// TwinCAT 3 PLC project lcls_plc_lps_02
// Title: lcls-plc-pls-02
// Company: SLAC
// ProjectVersion: 1.0.0
// ProgramVersion: 3.1.4022.7
// libraries:
//   Tc2_BABasic, * (Beckhoff Automation GmbH)
//   Tc2_EtherCAT, * (Beckhoff Automation GmbH)
//   Tc2_ModbusRTU, * (Beckhoff Automation GmbH)
//   Tc2_Standard, * (Beckhoff Automation GmbH)
//   Tc2_System, * (Beckhoff Automation GmbH)
//   Tc3_Module, * (Beckhoff Automation GmbH)
// project tree:
//   DUTs/ E_ShutterState.TcDUT, E_DeviceState.TcDUT, E_Mode.TcDUT, E_LeakLocation.TcDUT, ST_DeviceDiagnostic.TcDUT, ST_ErrorStates.TcDUT, ST_LaserSetpoints.TcDUT, ST_LeakBoundaries.TcDUT, ST_TemperatureMonitorSetpoints.TcDUT
//   GVLs/ GVL_EL3174.TcGVL, GVL_IO.TcGVL, GVL_Laser.TcGVL, GVL_PLC.TcGVL, GVL_TemperatureMonitor.TcGVL, GVL_TraceTek.TcGVL
//   / PlcTask.TcTTO
//   POUs/Communication/ FB_TraceTekModbus.TcPOU
//   POUs/Devices/ FB_BaseplateChiller.TcPOU, FB_Amphos_Enable.TcPOU, FB_ChillerLoop.TcPOU, FB_DumpChiller.TcPOU, FB_LaserInterlock.TcPOU, FB_Laser_Timer.TcPOU, FB_Laser_Timer_MPC.TcPOU, FB_LeakMonitor.TcPOU, FB_ShutterControl.TcPOU
//   POUs/Diagnostics/ FB_EcatDiag.TcPOU
//   POUs/Helpers/ FB_ErrorTriggers.TcPOU
//   POUs/Interlocks/ F_BaseplateChillerEnable.TcPOU, F_DumpChillerEnable.TcPOU
//   POUs/ MAIN.TcPOU
// real-time tasks:
//   TASK PlcTask: cycle T#10ms, priority 20, ADS port 350
// I/O:
//   DEVICE Device 1 (EtherCAT), AmsNetId 172.21.160.71.2.1
//     B950-231B-R03-DRL-01 (EK1200) [EK1200-5000 EtherCAT Power supply (2A E-Bus)]
//       EL3174_00_01 [EL3174 4Ch. Ana. Input +/-10V Diff., +/-20mA SingleEnded, 16 Bit]
//       EL3174_00_02 [EL3174 4Ch. Ana. Input +/-10V Diff., +/-20mA SingleEnded, 16 Bit]
//       EL9189_00_03 [EL9189 Potential Connection, 16 x Ground]
//       EL1259_00_04 [EL1259 8Ch. Dig Input 24V/8Ch. Dig. Output 24V with Multi-Time-Stamp]
//       EL9184_00_05 [EL9184 Potential Connection, 8 x 24V, 8 x Ground]
//       EL2624_00_07 [EL2624 4Ch. Relay Output, NO (125V AC / 30V DC)]
//       EL2624_00_08 [EL2624 4Ch. Relay Output, NO (125V AC / 30V DC)]
//       EL1004_00_8A
//       EL6022_00_09 [EL6022 Interface 2Ch. (RS422/485)]
//       EL9505_00_10
//       EL1124_00_11 [EL1124 4Ch. Dig. Input 5V, 10µs, Sensor Power]
//       EL1124_00_12
//       EL9011_00_12 [EL9011 End Terminal]
// variable links:
//   lcls_plc_lps_02 Instance <-> Device 1 (EtherCAT)/B950-231B-R03-DRL-01 (EK1200)/EL1004_00_8A
//     PlcTask Inputs/GVL_IO.bMirrorStatus <-> Channel 1/Input
//   lcls_plc_lps_02 Instance <-> Device 1 (EtherCAT)/B950-231B-R03-DRL-01 (EK1200)/EL1124_00_11
//     PlcTask Inputs/GVL_IO.bAmphosLaserReady <-> Channel 4/Input
//     PlcTask Inputs/GVL_IO.bAmphosOn <-> Channel 1/Input
//     PlcTask Inputs/GVL_IO.bAmphosShutterStatus <-> Channel 2/Input
//     PlcTask Inputs/GVL_IO.bCarbideOn <-> Channel 3/Input
//   lcls_plc_lps_02 Instance <-> Device 1 (EtherCAT)/B950-231B-R03-DRL-01 (EK1200)/EL1124_00_12
//     PlcTask Inputs/GVL_IO.bAmphosLaserACK <-> Channel 1/Input
//     PlcTask Inputs/GVL_IO.bAmphosLaserBusy <-> Channel 2/Input
//   lcls_plc_lps_02 Instance <-> Device 1 (EtherCAT)/B950-231B-R03-DRL-01 (EK1200)/EL1259_00_04
//     PlcTask Inputs/GVL_IO.bBaseplateChillerFlow <-> MTI Inputs 10x Channel 8/Status/Input state
//     PlcTask Inputs/GVL_IO.bDumpChillerFlow <-> MTI Inputs 10x Channel 7/Status/Input state
//     PlcTask Inputs/GVL_IO.bLoopTempSW01 <-> MTI Inputs 10x Channel 3/Status/Input state
//     PlcTask Inputs/GVL_IO.bLoopTempSW02 <-> MTI Inputs 10x Channel 4/Status/Input state
//     PlcTask Inputs/GVL_IO.bLoopTempSW03 <-> MTI Inputs 10x Channel 5/Status/Input state
//     PlcTask Inputs/GVL_IO.bLoopTempSW04 <-> MTI Inputs 10x Channel 6/Status/Input state
//     PlcTask Inputs/GVL_IO.bLoopTempSW05 <-> MTI Inputs 10x Channel 1/Status/Input state
//     PlcTask Inputs/GVL_IO.bTracetekAlarm <-> MTI Inputs 10x Channel 2/Status/Input state
//   lcls_plc_lps_02 Instance <-> Device 1 (EtherCAT)/B950-231B-R03-DRL-01 (EK1200)/EL2624_00_07
//     PlcTask Outputs/GVL_IO.bAmphosEnable <-> Channel 3/Output
//     PlcTask Outputs/GVL_IO.bBaseplateChillerRelay <-> Channel 2/Output
//     PlcTask Outputs/GVL_IO.bCarbideShutterEnable <-> Channel 4/Output
//     PlcTask Outputs/GVL_IO.bDumpChillerRelay <-> Channel 1/Output
//   lcls_plc_lps_02 Instance <-> Device 1 (EtherCAT)/B950-231B-R03-DRL-01 (EK1200)/EL2624_00_08
//     PlcTask Outputs/GVL_IO.bAmphosRelayCLOSE <-> Channel 4/Output
//     PlcTask Outputs/GVL_IO.bAmphosRelayOPEN <-> Channel 1/Output
//   lcls_plc_lps_02 Instance <-> Device 1 (EtherCAT)/B950-231B-R03-DRL-01 (EK1200)/EL3174_00_01
//     PlcTask Inputs/GVL_IO.nMultiPassVoltageRaw <-> AI Standard Channel 3/Value
//     PlcTask Inputs/GVL_IO.nOpcpaVoltageRaw <-> AI Standard Channel 1/Value
//   lcls_plc_lps_02 Instance <-> Device 1 (EtherCAT)/B950-231B-R03-DRL-01 (EK1200)/EL3174_00_02
//     PlcTask Inputs/GVL_IO.nAmphosVoltageRaw <-> AI Standard Channel 1/Value
//   lcls_plc_lps_02 Instance <-> Device 1 (EtherCAT)/B950-231B-R03-DRL-01 (EK1200)/EL6022_00_09
//     PlcTask Inputs/MAIN.fbTraceTekModbus.fbModbusMaster.InData/D <-> COM Inputs Channel 2/Data In 0
//     PlcTask Inputs/MAIN.fbTraceTekModbus.fbModbusMaster.InData/D @bit {8..168 step 8} <-> COM Inputs Channel 2/Data In {1..21}  (21 links)
//     PlcTask Inputs/MAIN.fbTraceTekModbus.fbModbusMaster.InData/Status <-> COM Inputs Channel 2/Status
//     PlcTask Outputs/MAIN.fbTraceTekModbus.fbModbusMaster.OutData/Ctrl <-> COM Outputs Channel 2/Ctrl
//     PlcTask Outputs/MAIN.fbTraceTekModbus.fbModbusMaster.OutData/D <-> COM Outputs Channel 2/Data Out 0
//     PlcTask Outputs/MAIN.fbTraceTekModbus.fbModbusMaster.OutData/D @bit {8..168 step 8} <-> COM Outputs Channel 2/Data Out {1..21}  (21 links)

CONFIGURATION lcls_plc_lps_02
    RESOURCE PLC ON TwinCAT3
        TASK PlcTask(INTERVAL := T#10ms, PRIORITY := 20);
        PROGRAM MAIN WITH PlcTask : MAIN;
    END_RESOURCE
END_CONFIGURATION

// ---- DUTs/E_ShutterState.TcDUT
{attribute 'qualified_only'}
{attribute 'strict'}
TYPE E_ShutterState :
(
    INIT := 0 ,
    OPENREQ := 1,
    OPENACK := 2,
    OPENTOGGLE := 3,
    OPENREADY:= 4,
    OPENED := 5,
    CLOSEREQ := 6,
    CLOSEACK := 7,
    CLOSETOGGLE := 8,
    CLOSEREADY := 9,
    CLOSED := 10,
    AMPHOSOFF := 11
);
END_TYPE

// ---- DUTs/E_DeviceState.TcDUT
{attribute 'qualified_only'}
TYPE E_DeviceState :
(
    INVALID := 0,
    INIT := EC_DEVICE_STATE_INIT,
    PREOP := EC_DEVICE_STATE_PREOP,
    BOOTSTRAP := EC_DEVICE_STATE_BOOTSTRAP,
    SAFEOP := EC_DEVICE_STATE_SAFEOP,
    OP := EC_DEVICE_STATE_OP
) WORD := INVALID;
END_TYPE

// ---- DUTs/E_Mode.TcDUT
{attribute 'qualified_only'}
TYPE E_Mode :
(
    MASTER_Override :=1,
    Protection := 2,
    AMPHOS_Maintenance := 3
);
END_TYPE

// ---- DUTs/E_LeakLocation.TcDUT
{attribute 'qualified_only'}
{attribute 'strict'}
TYPE E_LeakLocation :
(
    NO_LEAK := 0,
    LOC1 := 1,
    LOC2 := 2,
    LOC3 := 4,
    LOC4 := 8,
    LOC5 := 16,
    LOC6 := 32
) BYTE;
END_TYPE

// ---- DUTs/ST_DeviceDiagnostic.TcDUT
// PLC Terminal device diagnostics
TYPE ST_DeviceDiagnostic :
STRUCT
    {attribute 'pytmc' := '
        pv: TYPE
        io: i
    '}
    sType : STRING[15];
    {attribute 'pytmc' := '
        pv: ADDRESS
        io: i
    '}
    nAddr : WORD;
    {attribute 'pytmc' := '
        pv: NAME
        io: i
    '}
    sName : STRING[31];
    {attribute 'pytmc' := '
        pv: DEVICE_STATE
        io: i
        field: ZRVL 0
        field: ONVL 1
        field: TWVL 2
        field: THVL 3
        field: FRVL 4
        field: SXVL	8
        field: ZRST INVALID
        field: ONST INIT
        field: TWST PREOP
        field: THST BOOTSTRAP
        field: FRST SAFEOP
        field: SXST OP
        field: ZRSV MAJOR
        field: ONSV MAJOR
        field: TWSV MAJOR
        field: THSV MAJOR
        field: FRSV MAJOR
        field: FVSV MINOR
        field: SXSV NO_ALARM
        field: UNSV MAJOR
    '}
    nDeviceState : ENUM;
    {attribute 'pytmc' := '
        pv: DEVICE_STATE_FLAGS
        io: i
    '}
    nDeviceStateFlags : BYTE;
    {attribute 'pytmc' := '
        pv: LINK_STATE_FLAGS
        io: i
    '}
    nLinkStateFlags : BYTE;
END_STRUCT
END_TYPE

// ---- DUTs/ST_ErrorStates.TcDUT
// Error states that can occur in the program
TYPE ST_ErrorStates :
STRUCT
    // Leak Alarms
    bLeakOpticalTableAmphosOn : BOOL; // Leak on the optical table with Amphos on
    bLeakOpticalTableNoLaser : BOOL; // Leak on the optical table with no laser on
    bLeakOpcpaCarbideOn : BOOL; // Leak inside the OPCPA with Carbide on
    bLeakUnderTable : BOOL; // Leak under the table
    bLeakInsideRacks : BOOL; // Leak inside the racks

   // Temperature loop alarms
    bChillerLoop01 : BOOL; // Temperature too high in loop 01
    bChillerLoop02 : BOOL; // Temperature too high in loop 02
    bChillerLoop03 : BOOL; // Temperature too high in loop 03
    bChillerLoop04 : BOOL; // Temperature too high in loop 04
    bChillerLoop05 : BOOL; // Temperature too high in loop 05

    // Beam Errors
    bAmphosBeam : BOOL; // Amphos beam error
    bOpcpaBeam : BOOL; // OPCPA beam error
    bMPCBeam :BOOL;    // MPC beam error

    // Temperature monitors
    bTempMon01 : BOOL; // Temperature too high at location 01
    bTempMon02 : BOOL; // Temperature too high at location 02
    bTempMon03 : BOOL; // Temperature too high at location 03
    bTempMon04 : BOOL; // Temperature too high at location 04
    bTempMon05 : BOOL; // Temperature too high at location 05
    bTempMon06 : BOOL; // Temperature too high at location 06
    bTempMon07 : BOOL; // Temperature too high at location 07
    bTempMon08 : BOOL; // Temperature too high at location 08


    // Dump chiller
    bDumpChiller : BOOL; // Dump chiller error
    bBaseplateChiller : BOOL; // Baseplate chiller error

    // Hardware Failure
    bHardwareFailure : BOOL; // A component of the EPS has failed

    //Amphos Relay
    bAmphosRelay : BOOL; // Amphos Enable error

END_STRUCT
END_TYPE

// ---- DUTs/ST_LaserSetpoints.TcDUT
// Setpoints for the lasers
TYPE ST_LaserSetpoints :
STRUCT
    {attribute 'pytmc' := '
        pv: MIN_VOLTAGE
        io: io
        field: EGU Volts
    '}
    nMinVoltage : LREAL; // Minimum voltage the laser will be allowed to operate at
    {attribute 'pytmc' := '
        pv: MIN_NOMINAL_VOLTAGE
        io: io
        field: EGU Volts
    '}
    nMinNominalVoltage : LREAL; // Minimum voltage for the laser to be operating nominally
END_STRUCT
END_TYPE

// ---- DUTs/ST_LeakBoundaries.TcDUT
// Boundaries indicating leak monitor locations
TYPE ST_LeakBoundaries :
STRUCT
    {attribute 'pytmc' := '
        pv: L_MIN01
        io: io
    '}
    nLMin1 : UINT;
    {attribute 'pytmc' := '
        pv: L_MAX01
        io: io
    '}
    nLMax1 : UINT;
    {attribute 'pytmc' := '
        pv: L_MIN02
        io: io
    '}
    nLMin2 : UINT;
    {attribute 'pytmc' := '
        pv: L_MAX02
        io: io
    '}
    nLMax2 : UINT;
    {attribute 'pytmc' := '
        pv: L_MIN03
        io: io
    '}
    nLMin3 : UINT;
    {attribute 'pytmc' := '
        pv: L_MAX03
        io: io
    '}
    nLMax3 : UINT;
    {attribute 'pytmc' := '
        pv: L_MIN04
        io: io
    '}
    nLMin4 : UINT;
    {attribute 'pytmc' := '
        pv: L_MAX04
        io: io
    '}
    nLMax4 : UINT;
    {attribute 'pytmc' := '
        pv: L_MIN05
        io: io
    '}
    nLMin5 : UINT;
    {attribute 'pytmc' := '
        pv: L_MAX05
        io: io
    '}
    nLMax5 : UINT;
    {attribute 'pytmc' := '
        pv: L_MIN06
        io: io
    '}
    nLMin6 : UINT;
    {attribute 'pytmc' := '
        pv: L_MAX06
        io: io
    '}
    nLMax6 : UINT;
END_STRUCT
END_TYPE

// ---- DUTs/ST_TemperatureMonitorSetpoints.TcDUT
// Setpoints for the temperature monitors
TYPE ST_TemperatureMonitorSetpoints :
STRUCT
    {attribute 'pytmc' := '
        pv: MAX_TEMP
        io: io
        field: EGU C
    '}
    fMaxTemperature : LREAL; // Maximum temperature in Celsius allowed before triggering error
END_STRUCT
END_TYPE

// ---- GVLs/GVL_EL3174.TcGVL
{attribute 'qualified_only'}
VAR_GLOBAL CONSTANT
    (* Analog scaling *)
    fRawUpperLimit : LREAL := 16#7736; // Highest raw signal that can be read
    fRawLowerLimit : LREAL := 16#0000; // Lowest raw signal that can be read
    fScaleUpperLimit : LREAL := 10; // Upper limit in volts
    fScaleLowerLimit : LREAL := 0; // Lower limit in volts
END_VAR

// ---- GVLs/GVL_IO.TcGVL
// PLC IO from terminal modules
{attribute 'qualified_only'}
VAR_GLOBAL

    (* Slot1 EL3174 *)
    {attribute 'TcLinkTo' :=    'TIIB[EL3174_00_01]^AI Standard Channel 1^Value'}
    nOpcpaVoltageRaw AT %I* : INT; // Ch1 OPCPA Laser

    {attribute 'TcLinkTo' :=    'TIIB[EL3174_00_02]^AI Standard Channel 1^Value'}
    nAmphosVoltageRaw AT %I* : INT; // Ch2 Amphos Laser

    {attribute 'TcLinkTo' :=    'TIIB[EL3174_00_01]^AI Standard Channel 3^Value'}
    nMultiPassVoltageRaw AT %I* : INT; // Ch3 MultiPass Cell

 (* Slot4 EL1259 Inputs *)
    {attribute 'TcLinkTo' := 'TIIB[EL1259_00_04]^MTI Inputs 10x Channel 2^Status^Input state'}
    bTracetekAlarm AT %I* : BOOL; // Tracetek Alarm
    {attribute 'TcLinkTo' := 'TIIB[EL1259_00_04]^MTI Inputs 10x Channel 3^Status^Input state'}
    bLoopTempSW01 AT %I* : BOOL; // Ch3 Loop 01 NC Temp switch
    {attribute 'TcLinkTo' := 'TIIB[EL1259_00_04]^MTI Inputs 10x Channel 4^Status^Input state'}
    bLoopTempSW02 AT %I* : BOOL; // Ch4 Loop 02 NC Temp switch
    {attribute 'TcLinkTo' := 'TIIB[EL1259_00_04]^MTI Inputs 10x Channel 5^Status^Input state'}
    bLoopTempSW03 AT %I* : BOOL; // Ch5 Loop 03 NC Temp switch
    {attribute 'TcLinkTo' := 'TIIB[EL1259_00_04]^MTI Inputs 10x Channel 6^Status^Input state'}
    bLoopTempSW04 AT %I* : BOOL; // Ch6 Loop 04 NC Temp switch
    {attribute 'TcLinkTo' := 'TIIB[EL1259_00_04]^MTI Inputs 10x Channel 1^Status^Input state'}
    bLoopTempSW05 AT %I* : BOOL; // Ch1 Loop 05 NC Temp switch
    {attribute 'TcLinkTo' := 'TIIB[EL1259_00_04]^MTI Inputs 10x Channel 8^Status^Input state'}
    bBaseplateChillerFlow AT %I* : BOOL; // Baseplate chiller NC flow sensor
    {attribute 'TcLinkTo' := 'TIIB[EL1259_00_04]^MTI Inputs 10x Channel 7^Status^Input state'}
    bDumpChillerFlow AT %I* : BOOL; //Dump Chiller flow sensor

//LabJack IO connection Amphos controller TBD

    {attribute 'pytmc' := '
        pv: @(PREFIX):LPS:AMPHOS:POWER_STATE
        io: i
        field: ZNAM "OFF"
        field: ONAM "ON"
    '}
    {attribute 'TcLinkTo' := 'TIIB[EL1124_00_11]^Channel 1^Input'}
    bAmphosOn AT %I* : BOOL; //  Laser ON - LabJACK IO

    {attribute 'pytmc' := '
        pv: @(PREFIX):LPS:AMPHOS:LASER_READY
        io: i
        field: ZNAM "OFF"
        field: ONAM "ON"
    '}
    {attribute 'TcLinkTo' := 'TIIB[EL1124_00_11]^Channel 4^Input'}
    bAmphosLaserReady AT %I* : BOOL; //  Laser Ready - LabJACK IO

    {attribute 'pytmc' := '
        pv: @(PREFIX):LPS:AMPHOS:LASER_ACK
        io: i
        field: ZNAM "OFF"
        field: ONAM "ON"
    '}
    {attribute 'TcLinkTo' := 'TIIB[EL1124_00_12]^Channel 1^Input'}
    bAmphosLaserACK AT %I* : BOOL; //  Laser Acknowledge - LabJACK IO

    {attribute 'pytmc' := '
        pv: @(PREFIX):LPS:AMPHOS:LASER_BUSY
        io: i
        field: ZNAM "OFF"
        field: ONAM "ON"
    '}
    {attribute 'TcLinkTo' := 'TIIB[EL1124_00_12]^Channel 2^Input'}
    bAmphosLaserBusy AT %I* : BOOL; //  Laser Busy - LabJACK IO

    {attribute 'pytmc' := '
        pv: @(PREFIX):LPS:AMPHOS:SHUTTER_CMD
        io: io
        field: ZNAM "OFF"
        field: ONAM "ON"
    '}
    bAmphosShutterCMD : BOOL ; // CMD to Amphos for Shutter Operation

    {attribute 'pytmc' := '
        pv: @(PREFIX):LPS:AMPHOS:SHUTTER_ENABLE
        io: io
        field: ZNAM "OFF"
        field: ONAM "ON"
    '}
    bAmphosShutterEnable : BOOL; // Shutter Enable RBV from User

// Amphos Enable
     {attribute 'pytmc' := '
        pv: @(PREFIX):LPS:AMPHOS:ENABLE
        io: i
        field: OSV NO_ALARM
        field: ZSV MAJOR
        field: ZNAM DISABLED
        field: ONAM ENABLED
    '}
    {attribute 'TcLinkTo' := 'TIIB[EL2624_00_07]^Channel 3^Output'}
    bAmphosEnable AT %Q* : BOOL; // Amphos Override Relay

//LabJack IO Controls
    {attribute 'pytmc' := '
        pv: @(PREFIX):LPS:AMPHOS_SHUTTER:ENABLE
        io: i
        field: OSV NO_ALARM
        field: ZSV MAJOR
        field: ZNAM DISABLED
        field: ONAM ENABLED
    '}
    {attribute 'TcLinkTo' := 'TIIB[EL1124_00_11]^Channel 2^Input'}
    bAmphosShutterStatus AT %I* : BOOL; // EL1124_02 - Ch2 Labjack IO Amphos Shutter Status
    bAmphosShutterEnableManualOperation AT %Q* : BOOL := TRUE;

    {attribute 'pytmc' := '
        pv: @(PREFIX):LPS:AMPHOS_RELAY:ENABLE
        io: i
        field: OSV NO_ALARM
        field: ZSV MAJOR
        field: ZNAM DISABLED
        field: ONAM ENABLED
    '}
    {attribute 'TcLinkTo' := 'TIIB[EL2624_00_08]^Channel 1^Output'}
    bAmphosRelayOPEN AT %Q* : BOOL; // Labjack IO - Amphos CMD Shutter Open

    {attribute 'TcLinkTo' := 'TIIB[EL2624_00_08]^Channel 4^Output'}
    bAmphosRelayCLOSE AT %Q* : BOOL; // Labjack IO - Amphos CMD Shutter Close

//Carbide control
    {attribute 'pytmc' := '
        pv: @(PREFIX):LPS:CARBIDE_SHUTTER:ENABLE
        io: i
        field: OSV NO_ALARM
        field: ZSV MAJOR
        field: ZNAM DISABLED
        field: ONAM ENABLED
    '}
    {attribute 'TcLinkTo' := 'TIIB[EL2624_00_07]^Channel 4^Output'}
    bCarbideShutterEnable AT %Q* : BOOL; // Carbide Shutter Enable Relay
    bCarbideShutterEnableManualOperation AT %Q* : BOOL := TRUE;

    (* Slot11 EL1124 *)
    {attribute 'pytmc' := '
        pv: @(PREFIX):LPS:MPC:POWER_STATE
        io: i
        field: ZNAM "OFF"
        field: ONAM "ON"
    '}
    {attribute 'TcLinkTo' := 'TIIB[EL1124_00_11]^Channel 3^Input'}
    bCarbideOn AT %I* : BOOL; // Carbide RA Ready Signal

//Dump Chiller control
   {attribute 'pytmc' := '
        pv: @(PREFIX):LPS:DUMP_CHILLER_RELAY:ENABLE
        io: i
        field: OSV NO_ALARM
        field: ZSV MAJOR
        field: ZNAM DISABLED
        field: ONAM ENABLED
    '}
    {attribute 'TcLinkTo' := 'TIIB[EL2624_00_07]^Channel 1^Output'}
    bDumpChillerRelay AT %Q* : BOOL; // Ch1 Dump chiller NC relay
// Baseplate Chiller control
    {attribute 'pytmc' := '
        pv: @(PREFIX):LPS:BASEPLATE_CHILLER_RELAY:ENABLE
        io: i
        field: OSV NO_ALARM
        field: ZSV MAJOR
        field: ZNAM DISABLED
        field: ONAM ENABLED
    '}
    {attribute 'TcLinkTo' := 'TIIB[EL2624_00_07]^Channel 2^Output'}
    bBaseplateChillerRelay AT %Q* : BOOL; // Ch2 Baseplate chiller NC relay

// LSS Mirror Status
    {attribute 'pytmc' := '
        pv: @(PREFIX):LPS:MIRROR_STATUS
        io: i
        field: ZNAM "OFF"
        field: ONAM "ON"
    '}
    {attribute 'TcLinkTo' := 'TIIB[EL1004_00_8A]^Channel 1^Input'}
    bMirrorStatus AT %I* : BOOL; //  LSS Mirror Status

END_VAR

// ---- GVLs/GVL_Laser.TcGVL
// Setpoints for lasers
{attribute 'qualified_only'}
VAR_GLOBAL PERSISTENT
    {attribute 'pytmc' := 'pv: @(PREFIX):LPS:AMPHOS'}
    stAmphosSP : ST_LaserSetpoints; // Amphos setpoints
    {attribute 'pytmc' := 'pv: @(PREFIX):LPS:OPCPA'}
    stOpcpaSP : ST_LaserSetpoints; // OPCPA setpoints
    {attribute 'pytmc' := 'pv: @(PREFIX):LPS:MPC'}
    stMPCSP : ST_LaserSetpoints; // OPCPA setpoints
END_VAR

// ---- GVLs/GVL_PLC.TcGVL
// PLC global variables
{attribute 'qualified_only'}
VAR_GLOBAL
    AMSNetId AT %I* : AMSNETID;
END_VAR

// ---- GVLs/GVL_TemperatureMonitor.TcGVL
// Temperature monitor setpoints
{attribute 'qualified_only'}
VAR_GLOBAL PERSISTENT
    {attribute 'pytmc' := 'pv: @(PREFIX):LPS:TEMPMON01'}
    stTempMonSP01 : ST_TemperatureMonitorSetpoints;
    {attribute 'pytmc' := 'pv: @(PREFIX):LPS:TEMPMON02'}
    stTempMonSP02 : ST_TemperatureMonitorSetpoints;
    {attribute 'pytmc' := 'pv: @(PREFIX):LPS:TEMPMON03'}
    stTempMonSP03 : ST_TemperatureMonitorSetpoints;
    {attribute 'pytmc' := 'pv: @(PREFIX):LPS:TEMPMON04'}
    stTempMonSP04 : ST_TemperatureMonitorSetpoints;
    {attribute 'pytmc' := 'pv: @(PREFIX):LPS:TEMPMON05'}
    stTempMonSP05 : ST_TemperatureMonitorSetpoints;
    {attribute 'pytmc' := 'pv: @(PREFIX):LPS:TEMPMON06'}
    stTempMonSP06 : ST_TemperatureMonitorSetpoints;
    {attribute 'pytmc' := 'pv: @(PREFIX):LPS:TEMPMON07'}
    stTempMonSP07 : ST_TemperatureMonitorSetpoints;
    {attribute 'pytmc' := 'pv: @(PREFIX):LPS:TEMPMON08'}
    stTempMonSP08 : ST_TemperatureMonitorSetpoints;
END_VAR

// ---- GVLs/GVL_TraceTek.TcGVL
// Global variables for the TraceTek leak detector
{attribute 'qualified_only'}
VAR_GLOBAL CONSTANT
    (* Modbus address *)
    nModbusSlaveAddress : BYTE := 199; // Modbus slave address of the TraceTek device
END_VAR
VAR_GLOBAL PERSISTENT
    {attribute 'pytmc' := 'pv: @(PREFIX):LPS:LEAK'}
    stLeakMonitorBoundaries : ST_LeakBoundaries; // Boundaries of possible leak locations
END_VAR

// ---- POUs/MAIN.TcPOU
PROGRAM MAIN
VAR
    stErrors : ST_ErrorStates; // Triggered error states
    fbErrorTriggers : FB_ErrorTriggers; // Brand new errors this cycle

    // Leak Monitor
    {attribute 'pytmc' := 'pv: @(PREFIX):TTSIM:DEV01'}
    fbTraceTekModbus : FB_TraceTekModbus; // Modbus connection to TraceTek
    {attribute 'pytmc' := 'pv: @(PREFIX):LPS:LEAK:RESET'}
    bLeakMonitorReset : BOOL; // Leak monitor reset flag
    {attribute 'pytmc' := 'pv: @(PREFIX):LPS:LEAK'}
    fbLeakMonitor : FB_LeakMonitor; // Leak detection

    // Chiller Loop temperature monitors
    {attribute 'pytmc' := 'pv: @(PREFIX):LPS:TEMP01'}
    fbChillerLoop01 : FB_ChillerLoop; // Chiller loop 01
    {attribute 'pytmc' := 'pv: @(PREFIX):LPS:TEMP02'}
    fbChillerLoop02 : FB_ChillerLoop; // Chiller loop 02
    {attribute 'pytmc' := 'pv: @(PREFIX):LPS:TEMP03'}
    fbChillerLoop03 : FB_ChillerLoop; // Chiller loop 03
    {attribute 'pytmc' := 'pv: @(PREFIX):LPS:TEMP04'}
    fbChillerLoop04 : FB_ChillerLoop; // Chiller loop 04
    {attribute 'pytmc' := 'pv: @(PREFIX):LPS:TEMP05'}
    fbChillerLoop05 : FB_ChillerLoop; // Chiller loop 05

    // Laser monitors
    {attribute 'pytmc' := 'pv: @(PREFIX):LPS:AMPHOS'}
    fbAmphos : FB_Laser_Timer; // Amphos laser
    {attribute 'pytmc' := '
        pv: @(PREFIX):LPS:AMPHOS:RESET
        io: o
    '}
    bAmphosReset : BOOL; // Amphos laser error unlatch flag
    {attribute 'pytmc' := 'pv: @(PREFIX):LPS:OPCPA'}
    fbOpcpa : FB_Laser_Timer_MPC; // OPCPA laser
    {attribute 'pytmc' := '
        pv: @(PREFIX):LPS:OPCPA:RESET
        io: o
    '}
    bOpcpaReset : BOOL; // OPCPA laser error unlatch flag
    {attribute 'pytmc' := 'pv: @(PREFIX):LPS:MPC'}
    fbMPC : FB_Laser_Timer_MPC; // MultiPass Cell
    {attribute 'pytmc' := '
        pv: @(PREFIX):LPS:MPC:RESET
        io: o
    '}
    bMPCReset : BOOL; // MPC laser error unlatch flag
    {attribute 'pytmc' := '
        pv: @(PREFIX):LPS:MPC_MODE:RESET
        io: o
    '}
    fbAmphosEnable_MPC : FB_Amphos_Enable; // Latch for Amphos enable in MPC mode
    // Chillers
    {attribute 'pytmc' := 'pv: @(PREFIX):LPS:DUMP_CHILLER'}
    fbDumpChiller : FB_DumpChiller; // Flow sensor monitor for the dump chiller

    {attribute 'pytmc' := '
        pv: @(PREFIX):LPS:DUMP_CHILLER:RESET
        io: o
    '}
    bDumpChillerReset : BOOL; // Dump chiller error unlatch flag

    {attribute 'pytmc' := 'pv: @(PREFIX):LPS:BASEPLATE_CHILLER'}
    fbBaseplateChiller : FB_BaseplateChiller; // Flow sensor monitor for the baseplate chiller
    {attribute 'pytmc' := '
        pv: @(PREFIX):LPS:BASEPLATE_CHILLER:RESET
        io: o
    '}
    bBaseplateChillerReset : BOOL; // Baseplate chiller error unlatch flag

    {attribute 'pytmc' := '
        pv: @(PREFIX):LPS:MASTER_OVERRIDE
        io: o
    '}
    bMasterOverride : BOOL; // Master override control for safety system.

    (*
    This is the map of the Mode Int to the defintion
    MODE = 1 ==> Master Override
    MODE = 2 ==> Protection
    MODE = 3 ==> Amphos Maintenance
    Any other mode is invalid.
    We can later convert this MODE into an ENUM
    *)
    {attribute 'pytmc' := '
        pv: @(PREFIX):LPS:MODE
        io: io
        field: NOBT 3
    '}
    Mode_LPS : E_Mode; // Mode Definition

    {attribute 'pytmc' := 'pv: @(PREFIX):LPS:PLC'}
    fbDiag : FB_EcatDiag; // Ethercat diagnostics

    Shutter_State_ENUM : E_ShutterState; // Shutter State ENUM
    fb_ShutterControl : FB_ShutterControl; // Shutter control function block

    {attribute 'pytmc' := '
        pv: @(PREFIX):LPS:MASTER_LATCH_RESET
        io: o
    '}
    bMasterLatchReset : BOOL; //Master release of latched error conditions
    bLatchStart : BOOL := FALSE; //Latch at start of loop.

    fbShutterEnableInterlocks : FB_LaserInterlock;
END_VAR

(*******************************************************************
        Update diagnostics. Check for hardware failures
*******************************************************************)
(* Check PLC hardware for failures *)
//fbDiag(AMSNetId := GVL_PLC.AMSNetId);
//stErrors.bHardwareFailure := (fbDiag.bError OR fbTraceTekModbus.bError);
stErrors.bHardwareFailure := FALSE;

(* Ensure master latch is TRUE for at least one full cycle of the PLC logic *)
IF bMasterLatchReset AND NOT bLatchStart THEN
    bLatchStart := TRUE;
END_IF

(*******************************************************************
Feed each device function block inputs from the PLC IO. Collect error states detected
by the function blocks into stErrors. These collected errors are then used later for
making decisions in the interlock logic.
*******************************************************************)
(* Detects leaks using the location resitance from the TraceTek *)
fbLeakMonitor(
              nLocationResistance       := fbTraceTekModbus.nLocationResistance,
              bAmphosOn                 := GVL_IO.bAmphosOn,
              bCarbideOn                := GVL_IO.bCarbideOn,
              bLeakDetected             := GVL_IO.bTracetekAlarm,
              stBound                   := GVL_TraceTek.stLeakMonitorBoundaries,
              bLeakOpticalTableAmphosOn  => stErrors.bLeakOpticalTableAmphosOn,
              bLeakOpticaltableNoLaser   => stErrors.bLeakOpticalTableNoLaser,
              bLeakOpcpaCarbideOn        => stErrors.bLeakOpcpaCarbideOn,
              bLeakUnderTable            => stErrors.bLeakUnderTable,
              bLeakInsideRacks           => stErrors.bLeakInsideRacks
);


(* Monitors for error events on chiller loop 1 *)
fbChillerLoop01(
                bLoopTempSW     := GVL_IO.bLoopTempSW01,
                bError           => stErrors.bChillerLoop01
);

(* Monitors for error events on chiller loop 2 *)
fbChillerLoop02(
                bLoopTempSW     := GVL_IO.bLoopTempSW02,
                bError           => stErrors.bChillerLoop02
);

(* Monitors for error events on chiller loop 3 *)
fbChillerLoop03(
                bLoopTempSW     := GVL_IO.bLoopTempSW03,
                bError           => stErrors.bChillerLoop03
);

(* Monitors for error events on chiller loop 4 *)
fbChillerLoop04(
                bLoopTempSW     := GVL_IO.bLoopTempSW04,
                bError           => stErrors.bChillerLoop04
);

(* Monitors for error events on chiller loop 5 *)
fbChillerLoop05(
                bLoopTempSW     := GVL_IO.bLoopTempSW05,
                bError           => stErrors.bChillerLoop05
);


(* Monitors the Amphos laser *)
fbAmphos(
    nVoltageRaw := GVL_IO.nAmphosVoltageRaw,
    bAmphosOn := GVL_IO.bAmphosOn,
    stSetpoints := GVL_Laser.stAmphosSP,
    bError => stErrors.bAmphosBeam,
    bMasterLatchReset := bMasterLatchReset
);

(* Monitors the OPCPA laser *)
fbOpcpa(
        nVoltageRaw         := GVL_IO.nOpcpaVoltageRaw,
        bCarbideOn          := GVL_IO.bCarbideOn,
        stSetpoints         := GVL_Laser.stOpcpaSP,
        bError               => stErrors.bOpcpaBeam,
        bMasterLatchReset   := bMasterLatchReset
);

(* Monitors the MPC laser *)
fbMPC(
      nVoltageRaw           := GVL_IO.nMultiPassVoltageRaw,
      bCarbideOn            := GVL_IO.bCarbideOn,
      stSetpoints           := GVL_Laser.stMPCSP,
      bError                 => stErrors.bMPCBeam,
      bMasterLatchReset     := bMasterLatchReset
);

//Flow sensor monitor for the beam dump chiller
fbDumpChiller(
              //bAmphosOn := GVL_IO.bAmphosOn,
              bDumpChillerFlow      := GVL_IO.bDumpChillerFlow,
              bError                 => stErrors.bDumpChiller,
              bMasterLatchReset     := bMasterLatchReset
);

(* Flow sensor monitor for the baseplate chiller *)
fbBaseplateChiller(
                    bBaseplateChillerFlow := GVL_IO.bBaseplateChillerFlow,
                    bError                 => stErrors.bBaseplateChiller,
                    bMasterLatchReset     := bMasterLatchReset
);

// Latch for Amphos Enable in MPC mode
fbAmphosEnable_MPC(
                    bMasterLatchReset := bMasterLatchReset,
                    Mode              := Mode_LPS,
                    fAmphosVoltage    := fbAmphos.fVoltage,
                    bError             => stErrors.bAmphosRelay,
                    stAmphosSetpoints := GVL_Laser.stAmphosSP,
                    stErrors          := stErrors );


(*******************************************************************
Now that each of the input signals have been checked and errors stored,
run the interlock logic.
*******************************************************************)
// Amphos Enable Latch

fbShutterEnableInterlocks(
    fOpcpaVoltage           := fbOpcpa.fVoltage, // The voltage of the OPCPA
    fAmphosVoltage          := fbAmphos.fVoltage, // The Amphos voltage
    fMpcVoltage             := fbMPC.fVoltage, // The MPC Voltage
    AmphosStatus            := GVL_IO.bAmphosOn, //Amphos Laser Shutter Status
    bLoopTempOverride01     := fbChillerLoop01.bOperatorOverride, // Whether the chiller loop error is overriden
    bLoopTempOverride02     := fbChillerLoop02.bOperatorOverride, // Whether the chiller loop error is overriden
    bLoopTempOverride03     := fbChillerLoop03.bOperatorOverride, // Whether the chiller loop error is overriden
    bLoopTempOverride04     := fbChillerLoop04.bOperatorOverride, // Whether the chiller loop error is overriden
    bLoopTempOverride05     := fbChillerLoop05.bOperatorOverride, // Whether the chiller loop error is overriden
//    ShutterStatus := GVL_IO.bAmphosShutterStatus,
    bAmphosShutter          := GVL_IO.bAmphosShutterCMD,
    Mode                    := Mode_LPS,
    stErrors                := stErrors,
    stOpcpaSetpoints        := GVL_Laser.stOpcpaSP,
    stAmphosSetpoints       := GVL_Laser.stAmphosSP,
    stMPCSetPoints          := GVL_Laser.stMPCSP,
    bCarbideShutter          => GVL_IO.bCarbideShutterEnable
);

// Function block for Shutter Control to Amphos Software
fb_ShutterControl(
    CMDShutterOPEN 	:= GVL_IO.bAmphosRelayOPEN,
    CMDShutterCLOSE := GVL_IO.bAmphosRelayCLOSE,
    LaserBusy       := GVL_IO.bAmphosLaserBusy,
    LaserAck        := GVL_IO.bAmphosLaserACK,
    LaserON         := GVL_IO.bAmphosOn,
    ShutterState    := GVL_IO.bAmphosShutterStatus,
    Mode            := Mode_LPS);

(* Enable Dump chiller if interlock logic passes *)
GVL_IO.bDumpChillerRelay := F_DumpChillerEnable(
                                                stErrors := stErrors,
                                                Mode := Mode_LPS
                                                //bMasterOverride := bMasterOverride
);

(* Enable Baseplate chiller if interlock logic passes *)
GVL_IO.bBaseplateChillerRelay := F_BaseplateChillerEnable(
                                                          stErrors := stErrors,
                                                          Mode := Mode_LPS
                                                          //bMasterOverride := bMasterOverride
);

(*******************************************************************
Safety related tasks have now been finished. Now try slower tasks such as
communicating with external hardware.
*******************************************************************)
(* Read from TraceTek hardware to get leak details. Errors are
handled later when diagnostics are run *)
fbTraceTekModbus(
                 nModbusSlaveAddress := GVL_TraceTek.nModbusSlaveAddress,
                 bLeakDetected := GVL_IO.bTracetekAlarm
);

(*******************************************************************
As per the specification, the reset PV is not checked until after the EPS has taken action.
Check the reset flags to see if they have been set and the errors can be unlatched.
*******************************************************************)
(* Check for rising-edge errors *)
fbErrorTriggers(stErrors := stErrors);
(*
(* Check for new leak errors *)
IF fbErrorTriggers.NewLeakError() THEN
    bLeakMonitorReset := FALSE; // If there is a new error turn off reset
ELSIF bLeakMonitorReset THEN
    // If there are no new errors and reset is on, reset the errors
    fbLeakMonitor.Reset();
    fbErrorTriggers.ResetLeakTriggers();
END_IF
*)
(* Check for new Amphos beam errors *)
IF fbErrorTriggers.stNewErrors.bAmphosBeam THEN
    bAmphosReset := FALSE; // If there is a new error turn off reset
ELSIF bAmphosReset THEN
    // If there are no new errors and reset is on, reset the errors
    fbAmphos.Reset();
    fbErrorTriggers.ResetAmphosTrigger();
END_IF

(* Check for new OPCPA errors *)
IF fbErrorTriggers.stNewErrors.bOpcpaBeam THEN
    bOpcpaReset := FALSE; // If there is a new error turn off reset
ELSIF bOpcpaReset THEN
    // If there are no new errors and reset is on, reset the errors
    fbOpcpa.Reset();
    fbErrorTriggers.ResetOpcpaTrigger();
END_IF

(* Check for new MPC errors *)
IF fbErrorTriggers.stNewErrors.bMPCBeam THEN
     bMPCReset := FALSE; // If there is a new error turn off reset
ELSIF bMPCReset THEN
    // If there are no new errors and reset is on, reset the errors
    fbMPC.Reset();
    fbErrorTriggers.ResetMPCTrigger();
END_IF

(* Check for new Beam Dump chiller errors *)
IF fbErrorTriggers.stNewErrors.bDumpChiller THEN
    bDumpChillerReset := FALSE; // If there is a new error turn off reset
ELSIF bDumpChillerReset THEN
    fbDumpChiller.Reset();
    fbErrorTriggers.ResetDumpChillerTrigger();
END_IF

(* Check for new Baseplate chiller errors *)
IF fbErrorTriggers.stNewErrors.bBaseplateChiller THEN
    bBaseplateChillerReset := FALSE; // If there is a new error turn off reset
ELSIF bBaseplateChillerReset THEN
    // If there are no new errors and reset is on, reset the errors
    fbBaseplateChiller.Reset();
    fbErrorTriggers.ResetBaseplateChillerTrigger();
END_IF

(* Remove Master Latch Reset after one scan *)
IF bMasterLatchReset AND bLatchStart THEN
    bMasterLatchReset := FALSE;
    bLatchStart := FALSE;
END_IF

END_PROGRAM

// ---- POUs/Helpers/FB_ErrorTriggers.TcPOU
// Detects rising-edge errors
FUNCTION_BLOCK FB_ErrorTriggers
VAR_INPUT
    nLeakLocations : BYTE;
END_VAR
VAR_IN_OUT CONSTANT
    stErrors : ST_ErrorStates; // Errors that have been detected
END_VAR
VAR_OUTPUT
    stNewErrors : St_ErrorStates; // Rising-edge errors
END_VAR
VAR
    // R_TRIG function blocks for detecting new errors
    fbLeakTrig : R_TRIG;
    fbLeakOpticalTableAmphosOnTrig : R_TRIG;
    fbLeakOpticalTableNoLaserTrig : R_TRIG;
    fbLeakOpcpaCarbideOnTrig : R_TRIG;
    fbLeakUnderTableTrig : R_TRIG;
    fbLeakInsideRacksTrig : R_TRIG;
    fbAmphosBeamTrig : R_TRIG;
    fbOpcpaBeamTrig : R_TRIG;
    fbMPCBeamTrig : R_TRIG;
    fbDumpChillerTrig : R_TRIG;
    fbBaseplateChillerTrig : R_TRIG;

END_VAR

fbLeakTrig(
    CLK := nLeakLocations <> E_LeakLocation.NO_LEAK,
);
fbLeakOpticalTableAmphosOnTrig(
    CLK := stErrors.bLeakOpticalTableAmphosOn,
    Q => stNewErrors.bLeakOpticalTableAmphosOn
);
fbLeakOpticalTableNoLaserTrig(
    CLK := stErrors.bLeakOpticalTableNoLaser,
    Q => stNewErrors.bLeakOpticalTableNoLaser
);
fbLeakOpcpaCarbideOnTrig(
    CLK := stErrors.bLeakOpcpaCarbideOn,
    Q => stNewErrors.bLeakOpcpaCarbideOn
);
fbLeakUnderTableTrig(
    CLK := stErrors.bLeakUnderTable,
    Q => stNewErrors.bLeakUnderTable
);
fbLeakInsideRacksTrig(
    CLK := stErrors.bLeakInsideRacks,
    Q => stNewErrors.bLeakInsideRacks
);

fbAmphosBeamTrig(
    CLK := stErrors.bAmphosBeam,
    Q => stNewErrors.bAmphosBeam
);
fbOpcpaBeamTrig(
    CLK := stErrors.bOpcpaBeam,
    Q => stNewErrors.bOpcpaBeam
);

fbMPCBeamTrig(
    CLK := stErrors.bMPCBeam,
    Q => stNewErrors.bMPCBeam
);

fbDumpChillerTrig(
    CLK := stErrors.bDumpChiller,
    Q => stNewErrors.bDumpChiller
);
fbBaseplateChillerTrig(
    CLK := stErrors.bBaseplateChiller,
    Q => stNewErrors.bBaseplateChiller
);

// Returns whether a rising-edge leak error has occured
METHOD NewLeakError : BOOL
VAR_INPUT
END_VAR
NewLeakError := fbLeakTrig.Q OR fbLeakOpticalTableAmphosOnTrig.Q OR fbLeakOpticalTableNoLaserTrig.Q OR fbLeakOpcpaCarbideOnTrig.Q OR fbLeakUnderTableTrig.Q OR fbLeakInsideRacksTrig.Q;
END_METHOD

// Reset latched amphos errors
METHOD ResetAmphosTrigger
VAR_INPUT
END_VAR
fbAmphosBeamTrig(
    CLK := FALSE,
    Q => stNewErrors.bAmphosBeam
);
END_METHOD

METHOD ResetBaseplateChillerTrigger
VAR_INPUT
END_VAR
fbBaseplateChillerTrig(
    CLK := FALSE,
    Q => stNewErrors.bBaseplateChiller
);
END_METHOD

METHOD ResetDumpChillerTrigger
VAR_INPUT
END_VAR
fbDumpChillerTrig(
    CLK := FALSE,
    Q => stNewErrors.bDumpChiller
);
END_METHOD

// Reset latched leak errors
METHOD ResetLeakTriggers
VAR_INPUT
END_VAR
fbLeakOpticalTableAmphosOnTrig(
    CLK := FALSE,
    Q => stNewErrors.bLeakOpticalTableAmphosOn
);
fbLeakOpticalTableNoLaserTrig(
    CLK := FALSE,
    Q => stNewErrors.bLeakOpticalTableNoLaser
);
fbLeakOpcpaCarbideOnTrig(
    CLK := FALSE,
    Q => stNewErrors.bLeakOpcpaCarbideOn
);
fbLeakUnderTableTrig(
    CLK := FALSE,
    Q => stNewErrors.bLeakUnderTable
);
fbLeakInsideRacksTrig(
    CLK := FALSE,
    Q => stNewErrors.bLeakInsideRacks
);
END_METHOD

METHOD ResetMPCTrigger
VAR_INPUT
END_VAR
fbMPCBeamTrig(
    CLK := FALSE,
    Q => stNewErrors.bOpcpaBeam
);
END_METHOD

// Reset latched OPCPA errors
METHOD ResetOpcpaTrigger
VAR_INPUT
END_VAR
fbOpcpaBeamTrig(
    CLK := FALSE,
    Q => stNewErrors.bOpcpaBeam
);
END_METHOD

END_FUNCTION_BLOCK

// ---- POUs/Communication/FB_TraceTekModbus.TcPOU
// Communicates with the TraceTek TTSIM-1A hardware over Modbus to get more information about a leak
FUNCTION_BLOCK FB_TraceTekModbus
VAR_INPUT
    nModbusSlaveAddress : BYTE; // Modbus address of slave to be read from
    bLeakDetected : BOOL; // Whether a leak has been detected
    bResetError : BOOL; // Reset signal for error
END_VAR
VAR_OUTPUT
    {attribute 'pytmc' := '
        pv: LOC_RES
        io: input
    '}
    nLocationResistance: UINT; // Resistance measured in the detection wire
    {attribute 'pytmc' := '
        pv: ERROR
        io: i
        field: OSV MAJOR
        field: ZSV NO_ALARM
        field: ZNAM OK
        field: ONAM ERROR
    '}
    bError : BOOL := FALSE; // Flag for Modbus communication errors
    nErrorId : MODBUS_ERRORS := MODBUS_ERRORS.MODBUSERROR_NO_ERROR; // Description of Modbus error
END_VAR
VAR
    aModbusBuffer : WORD := 16#FFFF;  // "Infinite" until real value is read from device
    fbModbusMaster : ModbusRtuMaster_KL6x22B := (
        Quantity := 1,
        MBAddr := 1,
        cbLength := SIZEOF(aModbusBuffer),
        pMemoryAddr := ADR(aModbusBuffer),
        Timeout := T#5S
    );
    fbPoll : TON := (PT := T#0S); // Poll rate for reading modbus. Start at 0 so that modbus is read on first call
END_VAR
VAR_STAT
    tPollRate : TIME := T#500MS;
END_VAR

// Advance poll rate timer
fbPoll(IN := TRUE);

// Update modbus status
fbModbusMaster.Execute := FALSE;
fbModbusMaster.ReadInputRegs();

IF bResetError THEN // Reset modbus error
    bError := FALSE;
    nErrorId := MODBUS_ERRORS.MODBUSERROR_NO_ERROR;
ELSIF fbModbusMaster.Error OR NOT fbModbusMaster.BUSY THEN
    // Allow fb error state to go back to normal by checking modbus error state after reading has finished
    bError := fbModbusMaster.Error;
    nErrorId := fbModbusMaster.ErrorId;
END_IF

(* If the modbus interface isn't busy and there is a leak, try reading
the leak location from the TraceTek. Even if there is no leak, maintain
the modbus connection by checking every few seconds using the fbPoll rate *)
IF NOT fbModbusMaster.BUSY AND (bLeakDetected OR fbPoll.Q) THEN
    fbPoll(IN := FALSE, PT := tPollRate);
    fbModbusMaster.UnitID := nModbusSlaveAddress;
    fbModbusMaster.Execute := TRUE;
    fbModbusMaster.ReadInputRegs();
END_IF

// Copy the location resitance from the buffer to the FB output
nLocationResistance := WORD_TO_UINT(aModbusBuffer);

END_FUNCTION_BLOCK

// ---- POUs/Devices/FB_LeakMonitor.TcPOU
// Detect leaks and leak locations
FUNCTION_BLOCK FB_LeakMonitor
VAR_INPUT
    bLeakDetected : BOOL; // Whether a leak was detected
    bAmphosOn : BOOL; // Whether the Amphos is on
    bCarbideOn : BOOL; // Whether the Carbide is on
    nLocationResistance: UINT; // Used for calculating the location of the leak
END_VAR
VAR_IN_OUT CONSTANT
    stBound : ST_LeakBoundaries; // Setpoints for calculating leak locations from location resistance
END_VAR
VAR_OUTPUT

    {attribute 'pytmc' := '
        pv: LOW_RES
        io: i
    '}
    bLowResistance : BOOL := FALSE;

    {attribute 'pytmc' := '
        pv: LEAKS
        io: i
    '}
    nLeakLocations : BYTE := E_LeakLocation.NO_LEAK; // Locations of leaks
    {attribute 'pytmc' := '
        pv: LOTAO_ERROR
        io: i
        field: OSV MAJOR
        field: ZSV NO_ALARM
        field: ZNAM OK
        field: ONAM ERROR
    '}
    bLeakOpticalTableAmphosOn : BOOL := FALSE; // Leak on the optical table with Amphos on
    {attribute 'pytmc' := '
        pv: LOTNL_ERROR
        io: i
        field: OSV MAJOR
        field: ZSV NO_ALARM
        field: ZNAM OK
        field: ONAM ERROR
    '}
    bLeakOpticalTableNoLaser : BOOL := FALSE; // Leak on the optical table with no laser on
    {attribute 'pytmc' := '
        pv: LOCO_ERROR
        io: i
        field: OSV MAJOR
        field: ZSV NO_ALARM
        field: ZNAM OK
        field: ONAM ERROR
    '}
    bLeakOpcpaCarbideOn : BOOL := FALSE; // Leak inside the OPCPA with Carbide on
    {attribute 'pytmc' := '
        pv: LUT_ERROR
        io: i
        field: OSV MAJOR
        field: ZSV NO_ALARM
        field: ZNAM OK
        field: ONAM ERROR
    '}
    bLeakUnderTable : BOOL := FALSE; // Leak under the table
    {attribute 'pytmc' := '
        pv: LIR_ERROR
        io: i
        field: OSV MAJOR
        field: ZSV NO_ALARM
        field: ZNAM OK
        field: ONAM ERROR
    '}
    bLeakInsideRacks : BOOL := FALSE; // Leak inside the racks
END_VAR

IF (nLocationResistance < 200) THEN
    bLowResistance := TRUE;
ELSE
    bLowResistance := FALSE;
END_IF

IF (bLeakDetected OR bLowResistance) THEN
    (* Find leak location for PV. Stays until reset *)
    IF stBound.nLMin1 <= nLocationResistance AND nLocationResistance < stBound.nLMax1 THEN
        nLeakLocations := nLeakLocations OR E_LeakLocation.LOC1;
    ELSIF stBound.nLMin2 <= nLocationResistance AND nLocationResistance < stBound.nLMax2 THEN
        nLeakLocations := nLeakLocations OR E_LeakLocation.LOC2;
    ELSIF stBound.nLMin3 <= nLocationResistance AND nLocationResistance < stBound.nLMax3 THEN
        nLeakLocations := nLeakLocations OR E_LeakLocation.LOC3;
    ELSIF stBound.nLMin4 <= nLocationResistance AND nLocationResistance < stBound.nLMax4 THEN
        nLeakLocations := nLeakLocations OR E_LeakLocation.LOC4;
    ELSIF stBound.nLMin5 <= nLocationResistance AND nLocationResistance < stBound.nLMax5 THEN
        nLeakLocations := nLeakLocations OR E_LeakLocation.LOC5;
    ELSIF stBound.nLMin6 <= nLocationResistance AND nLocationResistance < stBound.nLMax6 THEN
        nLeakLocations := nLeakLocations OR E_LeakLocation.LOC6;
    END_IF


    (* Latch Optical table leak errors *)
    IF (stBound.nLMin1 <= nLocationResistance AND nLocationResistance < stBound.nLMax4) THEN
        IF bAmphosOn THEN
            bLeakOpticalTableAmphosOn := TRUE;
        ELSIF NOT bCarbideOn THEN
            bLeakOpticalTableNoLaser := TRUE;
        END_IF
    END_IF

    (* Latch carbide leak errors *)
    IF (bCarbideOn AND stBound.nLMin1 <= nLocationResistance AND nLocationResistance < stBound.nLMax2) THEN
        bLeakOpcpaCarbideOn := TRUE;
    END_IF

    (* Latch leak under table errors *)
    IF (stBound.nLMin5 <= nLocationResistance AND nLocationResistance < stBound.nLMax5) THEN
        bLeakUnderTable := TRUE;
    END_IF

    (* Latch leak inside rack errors *)
    IF (stBound.nLMin6 <= nLocationResistance AND nLocationResistance < stBound.nLMax6) THEN
        bLeakInsideRacks := TRUE;
    END_IF
    (* Temp code*)
    IF bLeakDetected THEN
         bLeakUnderTable := TRUE;
         bLeakInsideRacks := TRUE;
    END_IF

END_IF

// Reset latched errors
METHOD Reset
VAR_INPUT
END_VAR
nLeakLocations := E_LeakLocation.NO_LEAK;
bLeakOpticalTableAmphosOn := FALSE;
bLeakOpticalTableNoLaser := FALSE;
bLeakOpcpaCarbideOn := FALSE;
bLeakUnderTable := FALSE;
bLeakInsideRacks := FALSE;
END_METHOD

END_FUNCTION_BLOCK

// ---- POUs/Devices/FB_ChillerLoop.TcPOU
// Monitors the chiller loop from the flow sensor
FUNCTION_BLOCK FB_ChillerLoop
VAR_INPUT
    bLoopTempSW : BOOL; // NC Temperature switch. Indicates when temperature is too high
END_VAR
VAR_OUTPUT
    {attribute 'pytmc' := '
        pv: ERROR
        io: i
        field: OSV MAJOR
        field: ZSV NO_ALARM
        field: ZNAM OK
        field: ONAM ERROR
    '}
    bError : BOOL := FALSE; // Whether an error was detected. Goes back to normal on its own
    {attribute 'pytmc' := '
        pv: OVERRIDE
        io: io
        field: ZNAM "OFF"
        field: ONAM "ON"
    '}
    bOperatorOverride : BOOL := FALSE; // If TRUE, allows the EPS to keep running despite the chiller loop error
END_VAR

(* Set error flag if loop temperature monitor detects an error *)
bError := NOT bLoopTempSW;

(* Reset the operator override if the system returns to normal tempreature range *)
IF bLoopTempSW THEN
    bOperatorOverride := FALSE;
END_IF

END_FUNCTION_BLOCK

// ---- POUs/Devices/FB_Laser_Timer.TcPOU
// Monitors the lasers for under voltage events
FUNCTION_BLOCK FB_Laser_Timer
VAR_INPUT
    nVoltageRaw : INT; // The raw signal collected from the ADC
    bAmphosOn : BOOL; // Whether the amphos is turned on
    Timer : TON ; //Timer for reset
    bMasterLatchReset : BOOL; //Master latched error reset
    bCarbideOn : BOOL; // Whether Carbide is ON
    Mode : E_Mode;
END_VAR
VAR_IN_OUT CONSTANT
    stSetpoints : ST_LaserSetpoints; // Setpoints for the laser
END_VAR
VAR_OUTPUT
    {attribute 'pytmc' := '
        pv: VOLTAGE
        io: i
        field: HOPR 10.0
        field: LOPR 0.0
        field: LSV MINOR
        field: LLSV MAJOR
        field: EGU Volts
    '}
    fVoltage : LREAL; // Voltage calculated from the raw ADC input

    {attribute 'pytmc' := '
        pv: SCALED_PWR
        io: i
        field: EGU Watts
    '}
    fPower : LREAL;

    {attribute 'pytmc' := '
        pv: ERROR
        io: i
        field: OSV MAJOR
        field: ZSV NO_ALARM
        field: ZNAM OK
        field: ONAM ERROR
    '}
    bError : BOOL; // Whether an error was detected. Latches until reset
    bBelowNominal : BOOL; //fVoltage is below the nominal setpoint
END_VAR

(* Scale the analog signal to voltage *)
fVoltage := F_Scale(
    fRawData := nVoltageRaw,
    fRawDataLowerOffLimit := GVL_EL3174.fRawLowerLimit,
    fRawDataUpperOffLimit := GVL_EL3174.fRawUpperLimit,
    fScaleDataLowerOffLimit := GVL_EL3174.fScaleLowerLimit,
    fScaleDataUpperOffLimit := GVL_EL3174.fScaleUpperLimit);

fPower := fVoltage; //Value is scaled by user set ASLO and AOFF fields (for display only)

(* Set error if amphos is below nominal voltage *)
IF  (bAmphosOn AND fVoltage < stSetpoints.nMinVoltage) THEN
    Timer(IN:=TRUE, PT:=T#500ms); //500ms SEC Timer
        IF Timer.Q THEN
            bError := TRUE;
            Timer(IN:=FALSE);
        END_IF;
ELSE
    Timer(IN:=FALSE);
END_IF

IF bAmphosOn AND (fVoltage < stSetpoints.nMinNominalVoltage) THEN
    bBelowNominal := TRUE;
END_IF

IF bMasterLatchReset THEN
    bBelowNominal := FALSE;
    bError := FALSE;
END_IF

// Reset latched errors
METHOD Reset
VAR_INPUT
END_VAR
bError := FALSE;
END_METHOD

END_FUNCTION_BLOCK

// ---- POUs/Devices/FB_Laser_Timer_MPC.TcPOU
// Monitors the lasers for under voltage events
FUNCTION_BLOCK FB_Laser_Timer_MPC
VAR_INPUT
    nVoltageRaw : INT; // The raw signal collected from the ADC
    bCarbideOn : BOOL; // Whether the amphos is turned on
    Timer : TON ; //Timer for reset
    bMasterLatchReset : BOOL; //Master latched error reset
END_VAR
VAR_IN_OUT CONSTANT
    stSetpoints : ST_LaserSetpoints; // Setpoints for the laser
END_VAR
VAR_OUTPUT
    {attribute 'pytmc' := '
        pv: VOLTAGE
        io: i
        field: HOPR 10.0
        field: LOPR 0.0
        field: LSV MINOR
        field: LLSV MAJOR
        field: EGU Volts
    '}
    fVoltage : LREAL; // Voltage calculated from the raw ADC input

    {attribute 'pytmc' := '
        pv: SCALED_PWR
        io: i
        field: EGU Watts
    '}
    fPower : LREAL;

    {attribute 'pytmc' := '
        pv: ERROR
        io: i
        field: OSV MAJOR
        field: ZSV NO_ALARM
        field: ZNAM OK
        field: ONAM ERROR
    '}
    bError : BOOL; // Whether an error was detected. Latches until reset
    bBelowNominal : BOOL; //fVoltage is below the nominal setpoint
END_VAR

(* Scale the analog signal to voltage *)
fVoltage := F_Scale(
    fRawData := nVoltageRaw,
    fRawDataLowerOffLimit := GVL_EL3174.fRawLowerLimit,
    fRawDataUpperOffLimit := GVL_EL3174.fRawUpperLimit,
    fScaleDataLowerOffLimit := GVL_EL3174.fScaleLowerLimit,
    fScaleDataUpperOffLimit := GVL_EL3174.fScaleUpperLimit);

fPower := fVoltage; //Value is scaled by user set ASLO and AOFF fields (for display only)

(* Set error if amphos is below nominal voltage *)
IF  (bCarbideOn AND fVoltage < stSetpoints.nMinVoltage) THEN
    Timer(IN:=TRUE, PT:=T#500ms); //1 SEC Timer
    IF Timer.Q THEN
    bError := TRUE;
    Timer(IN:=FALSE);   // Reset Timer
    END_IF;
ELSE
    Timer(IN:=FALSE);
END_IF

IF bCarbideOn AND (fVoltage < stSetpoints.nMinNominalVoltage) THEN
    bBelowNominal := TRUE;
END_IF

IF bMasterLatchReset THEN
    bBelowNominal := FALSE;
    bError := FALSE;
END_IF

// Reset latched errors
METHOD Reset
VAR_INPUT
END_VAR
bError := FALSE;
END_METHOD

END_FUNCTION_BLOCK

// ---- POUs/Devices/FB_Amphos_Enable.TcPOU
// Monitors the baseplate chiller from the flow sensor
FUNCTION_BLOCK FB_Amphos_Enable
VAR_INPUT
    //bAmphosOn         : BOOL; // Whether the amphos is turned on
    //bAmphosEnable      : BOOL; // Signal from the flow sensor. Normally high.
    bMasterLatchReset : BOOL; //Master latched error reset
    fAmphosVoltage    : LREAL; // The Amphos voltage
END_VAR

VAR_OUTPUT
    {attribute 'pytmc' := '
        pv: ERROR
        io: i
        field: OSV MAJOR
        field: ZSV NO_ALARM
        field: ZNAM OK
        field: ONAM ERROR
    '}
    bError            : BOOL; // Whether an error was detected. Should latch until reset
END_VAR

VAR_IN_OUT CONSTANT
    stErrors          : ST_ErrorStates; // Currently detected errors
   // stOpcpaSetpoints : ST_LaserSetpoints; // OPCPA setpoints
    stAmphosSetpoints : ST_LaserSetpoints; // The Amphos setpoints
END_VAR

VAR_IN_OUT
    Mode              : E_Mode; // Mode
END_VAR

VAR
END_VAR

(* Latch error if the baseplate chiller flow detects an error *)
CASE MODE OF
    E_Mode.MASTER_Override, E_Mode.Protection, E_Mode.AMPHOS_Maintenance:
    IF fAmphosVoltage < stAmphosSetpoints.nMinVoltage
        THEN
            bError := TRUE;
        ELSE
            bError := FALSE;
    END_IF
    // Undefined state, do not get here
    ELSE
        Mode := E_Mode.Protection;
END_CASE

IF bMasterLatchReset THEN
    bError := FALSE;
END_IF

// Reset latched errors
METHOD Reset
VAR_INPUT
END_VAR
bError := FALSE;
END_METHOD

END_FUNCTION_BLOCK

// ---- POUs/Devices/FB_DumpChiller.TcPOU
// Monitors the dump chiller from the flow sensor
FUNCTION_BLOCK FB_DumpChiller
VAR_INPUT
    //bAmphosOn : BOOL; // Whether the amphos is turned on
    bDumpChillerFlow : BOOL; // Signal from the flow sensor. Normally high.
    bMasterLatchReset : BOOL; //Master latched error reset
END_VAR
VAR_OUTPUT
    {attribute 'pytmc' := '
        pv: ERROR
        io: i
        field: OSV MAJOR
        field: ZSV NO_ALARM
        field: ZNAM OK
        field: ONAM ERROR
    '}
    bError : BOOL; // Whether an error was detected. Latches until reset
END_VAR
VAR
END_VAR

(* Latch error if the dump chiller flow detects an error and the amphos is on *)
IF (NOT bDumpChillerFlow) THEN
    bError := TRUE;
END_IF

IF bMasterLatchReset THEN
    bError := FALSE;
END_IF

// Reset latched errors
METHOD Reset
VAR_INPUT
END_VAR
bError := FALSE;
END_METHOD

END_FUNCTION_BLOCK

// ---- POUs/Devices/FB_BaseplateChiller.TcPOU
// Monitors the baseplate chiller from the flow sensor
FUNCTION_BLOCK FB_BaseplateChiller
VAR_INPUT
    //bAmphosOn : BOOL; // Whether the amphos is turned on
    bBaseplateChillerFlow : BOOL; // Signal from the flow sensor. Normally high.
    bMasterLatchReset : BOOL; //Master latched error reset
END_VAR
VAR_OUTPUT
    {attribute 'pytmc' := '
        pv: ERROR
        io: i
        field: OSV MAJOR
        field: ZSV NO_ALARM
        field: ZNAM OK
        field: ONAM ERROR
    '}
    bError : BOOL; // Whether an error was detected. Should latch until reset
END_VAR
VAR
END_VAR

(* Latch error if the baseplate chiller flow detects an error *)
IF ( NOT bBaseplateChillerFlow ) THEN
    bError := TRUE;
END_IF

IF bMasterLatchReset THEN
    bError := FALSE;
END_IF

// Reset latched errors
METHOD Reset
VAR_INPUT
END_VAR
bError := FALSE;
END_METHOD

END_FUNCTION_BLOCK

// ---- POUs/Diagnostics/FB_EcatDiag.TcPOU
(*
Ecat bus diagnostic tool
2015-11-4 Alex Wallace
This function block checks the states of all slaves on the ecat bus network,
it could be modified to export the states of the slaves on an individual basis,
but for now it sets the output boolean true if all slaves are OP and false otherwise.
To start the block provide a falling edge on the first pass boolean input.

2018-05-05 Margaret Ghaly
Function block has been modified to retrieve the Device State of the Ethercat Master.
It also exports the states and information of each individual configured Slave.
And saves them in the array q_aEcConfSlaveInfo.

2019-08-28 Nathan Telles
Customized for EPS project using PyTMC. Export all states to a structure which is
linked to EPICS records. Remove unecessary diagnostics.
*)
{attribute 'call_after_init'}
FUNCTION_BLOCK FB_EcatDiag
VAR_INPUT
    {attribute 'naming' := 'omit'}
    AMSNetId : AMSNETID; //Link to the AMSNETID name in the ethercat master info.
    //i_xFirstPass: BOOL; //Hook to system first pass boolean for proper intialization (must be true for the first cycle of the PLC)
END_VAR
VAR_OUTPUT
    {attribute 'pytmc' := '
        pv: ERROR
        io: i
        field: OSV MAJOR
        field: ZSV NO_ALARM
        field: ZNAM OK
        field: ONAM ERROR
    '}
    bError : BOOL;
    {attribute 'pytmc' := '
        pv: SLAVES_OK
        io: i
        field: OSV NO_ALARM
        field: ZSV MAJOR
        field: ZNAM ERROR
        field: ONAM OK
    '}
    bAllSlaveStatesGood: BOOL; // Set to True if all Slaves are in OP State
    {attribute 'pytmc' := '
        pv: MASTER_OK
        io: i
        field: OSV NO_ALARM
        field: ZSV MAJOR
        field: ZNAM ERROR
        field: ONAM OK
    '}
    bMasterStateGood : BOOL;
END_VAR
VAR
    {attribute 'pytmc' := '
        pv: MASTER_DEV_STATE
        io: i
    '}
    nMasterDevState: WORD; // The Device State of the Master
    {attribute 'pytmc' := '
        pv: MASTER_STATE
        io: i
    '}
    nMasterState: WORD; // The State of the Master
    {attribute 'pytmc' := '
        pv: AMS_ID
        io: i
    '}
    sNetId: STRING(23); //NetId string

    astTermStates: ARRAY[1..MAX_SLAVES] OF ST_EcSlaveState; //ECAT Slave States Buffer
    astEcConfSlaveInfo: ARRAY[1..MAX_SLAVES] OF ST_EcSlaveConfigData; //ECAT Slave Configs Buffer

    fbGetAllSlaveStates: FB_EcGetAllSlaveStates; //Acquires the ECAT Slave States puts them into astTermStates
    fbGetMasterDevState: FB_EcGetMasterDevState; //Acquires ECAT Master State
    fbGetMasterState: FB_EcGetMasterState; //Acquires ECAT Master State
    fbGetConfSlaves: FB_EcGetConfSlaves; //Acquires the ECAT slave configuration of the bus (how many, what kind, etc)

    {attribute 'naming' := 'omit'}
    ftReset: F_TRIG; //Reset trigger sensor
    {attribute 'naming' := 'omit'}
    ftMasterDevReset: F_TRIG; //Retrigger sensor for GetMasterDevState
    {attribute 'naming' := 'omit'}
    ftMasterReset: F_TRIG; //Retrigger sensor for GetMasterState

    {attribute 'pytmc' := 'pv: SLAVE01'}
    stSlave01 : ST_DeviceDiagnostic;
    {attribute 'pytmc' := 'pv: SLAVE02'}
    stSlave02 : ST_DeviceDiagnostic;
    {attribute 'pytmc' := 'pv: SLAVE03'}
    stSlave03 : ST_DeviceDiagnostic;
    {attribute 'pytmc' := 'pv: SLAVE04'}
    stSlave04 : ST_DeviceDiagnostic;
    {attribute 'pytmc' := 'pv: SLAVE05'}
    stSlave05 : ST_DeviceDiagnostic;
    {attribute 'pytmc' := 'pv: SLAVE06'}
    stSlave06 : ST_DeviceDiagnostic;
    {attribute 'pytmc' := 'pv: SLAVE07'}
    stSlave07 : ST_DeviceDiagnostic;
    {attribute 'pytmc' := 'pv: SLAVE08'}
    stSlave08 : ST_DeviceDiagnostic;
    {attribute 'pytmc' := 'pv: SLAVE09'}
    stSlave09 : ST_DeviceDiagnostic;
    {attribute 'pytmc' := 'pv: SLAVE10'}
    stSlave10 : ST_DeviceDiagnostic;

    aSlaves : ARRAY [1..MAX_SLAVES] OF POINTER TO ST_DeviceDiagnostic := [ADR(stSlave01),ADR(stSlave02),
        ADR(stSlave03),ADR(stSlave04),ADR(stSlave05),ADR(stSlave06),ADR(stSlave07),ADR(stSlave08),
        ADR(stSlave09), ADR(stSlave10)];

    nIterator: UINT;
    bInit : BOOL := TRUE;

    {attribute 'pytmc' := '
        pv: SLAVES_COUNT
        io: i
    '}
    nSlaves : UINT;
END_VAR
VAR CONSTANT
    MAX_SLAVES : UINT := 10;
END_VAR

sNetId := F_CreateAmsNetId(AMSNetId);

//Query the state of all terminals, collect in astTermStates
ftReset(CLK:=fbGetAllSlaveStates.bBusy OR bInit);
fbGetAllSlaveStates.bExecute := ftReset.Q;
fbGetAllSlaveStates(sNetId:=sNetId, pStateBuf := ADR(astTermStates), cbBufLen:=SIZEOF(astTermStates));
//Keep checking...


//Cycle through each entry in the array and check if we have anyone not in OP and that the link state is good.
// If so, then set our global IO bad boolean.
IF fbGetAllSlaveStates.nSlaves > 0 THEN
    bAllSlaveStatesGood := TRUE;
    FOR nIterator := 1 TO MAX_SLAVES DO
        IF nIterator > fbGetAllSlaveStates.nSlaves // Slave is missing
        OR NOT( (astTermStates[nIterator].deviceState = EC_DEVICE_STATE_OP) AND (astTermStates[nIterator].linkState = EC_LINK_STATE_OK))
        THEN
            bAllSlaveStatesGood := FALSE;
        END_IF

        IF nIterator <= fbGetAllSlaveStates.nSlaves THEN
            aSlaves[nIterator]^.nDeviceState := astTermStates[nIterator].deviceState AND EC_DEVICE_STATE_MASK;
            aSlaves[nIterator]^.nDeviceStateFlags := SHR(astTermStates[nIterator].deviceState, 4);
            aSlaves[nIterator]^.nLinkStateFlags :=astTermStates[nIterator].linkState;
        ELSE
            // Missing slaves should be set to invalid
            aSlaves[nIterator]^.nDeviceState := E_DeviceState.INVALID;
        END_IF
    END_FOR
END_IF

// Read the EtherCAT state of the master. If the call is successful,
//the State output variable of type WORD contains the requested status information.
ftMasterDevReset(CLK:=fbGetMasterDevState.bBusy OR bInit);
fbGetMasterDevState(sNetId:= sNetId, bExecute:=ftMasterDevReset.Q, nDevState => nMasterDevState);

ftMasterReset(CLK:=fbGetMasterState.bBusy OR bInit);
fbGetMasterState(sNetId:= sNetId, bExecute:=ftMasterDevReset.Q, state => nMasterState);

bMasterStateGood:= (fbGetMasterState.state = BYTE_TO_UINT(EC_DEVICE_STATE_OP) AND fbGetMasterDevState.nDevState = 0);

//This function is used to read a list of all configured slaves from the EtherCat master object Directory
//needs to run only once
fbGetConfSlaves(bExecute := bInit, sNetId :=sNetId, pArrEcConfSlaveInfo := ADR(astEcConfSlaveInfo),cbBufLen := SIZEOF(astEcConfSlaveInfo));
nSlaves:=fbGetConfSlaves.nSlaves;

IF  NOT (fbGetConfSlaves.bBusy) THEN
    FOR nIterator := 1 TO MIN(MAX_SLAVES, fbGetConfSlaves.nSlaves) DO
        IF nIterator > fbGetConfSlaves.nSlaves THEN // Missing terminal
            aSlaves[nIterator]^.nAddr := 0;
            aSlaves[nIterator]^.sName := '';
            aSlaves[nIterator]^.sType := '';
        ELSE
            aSlaves[nIterator]^.nAddr :=astEcConfSlaveInfo[nIterator].nAddr;
            aSlaves[nIterator]^.sName :=astEcConfSlaveInfo[nIterator].sName;
            aSlaves[nIterator]^.sType :=astEcConfSlaveInfo[nIterator].sType;
        END_IF
    END_FOR
    fbGetConfSlaves.bExecute := FALSE;
END_IF


bInit := FALSE;
bError := fbGetMasterDevState.bError OR fbGetMasterState.bError OR fbGetAllSlaveStates.bError OR
    fbGetConfSlaves.bError OR NOT bAllSlaveStatesGood OR NOT bMasterStateGood;

END_FUNCTION_BLOCK

// ---- POUs/Devices/FB_ShutterControl.TcPOU
FUNCTION_BLOCK FB_ShutterControl
VAR_INPUT
    CMDShutterOPEN : BOOL; 			// CMD Shutter OPEN Relay state current state from EL2624 Relay
    CMDShutterCLOSE : BOOL; 		// CMD Shutter CLOSE Relay state current state from EL2624 Relay
    LaserBusy : BOOL;				// Laser Busy bit from Labjack IO
    LaserAck : BOOL;				// Laser Acknowledge bit from Labjack IO
    ShutterState : BOOL;		  	// Shutter state from Labjack IO
    LaserON : BOOL; 				// Laser ON state from Labjack
    T_OPENREQ : TON ; 			//Timer for reset
    T_OPENTOG : TON; 			// Timer for OPEN Toggle
    T_CLOSEREQ : TON;
    T_CLOSETOG : TON;
    Interlock_bit : BOOL; 			// From function block
    Mode : E_Mode; 					//Mode Definition
END_VAR
VAR_OUTPUT
    State : E_ShutterState := 0; 	// ENUM States
END_VAR

/// Function to assess CMD shutter state to Amphos
/// Logic will follow the following
// GVL_IO.bAmphosShutterCMD := TRUE ( Request to OPEN Shutter)
// GVL_IO.bAmphosShutterCMD := FALSE( Request to CLOSE Shutter)
///// AMPHOS Shutter State Descriptions:
//////// TRUE : CLOSED
//////// FALSE : OPEN


CASE State OF

E_ShutterState.INIT :
    GVL_IO.bAmphosRelayOPEN := TRUE;
    GVL_IO.bAmphosRelayCLOSE := TRUE;
    IF ShutterState
    THEN
        State := E_ShutterState.CLOSED;
        ELSE
        State := E_ShutterState.OPENED;
    END_IF

E_ShutterState.AMPHOSOFF :
    IF GVL_IO.bAmphosOn THEN
    State := E_ShutterState.INIT;
    END_IF

E_ShutterState.OPENREQ :
    IF GVL_IO.bAmphosOn THEN
    GVL_IO.bAmphosRelayCLOSE := TRUE;
    GVL_IO.bAmphosRelayOPEN := FALSE;
        IF GVL_IO.bAmphosLaserACK OR (NOT ShutterState) THEN
        State := E_ShutterState.OPENACK;
        END_IF
    ELSE
    State := E_ShutterState.AMPHOSOFF;
    END_IF
(*
    IF GVL_IO.bAmphosShutterCMD AND ShutterState AND LaserON AND (NOT LaserBusy)
        THEN
        GVL_IO.bAmphosRelayOPEN := FALSE;
        GVL_IO.bAmphosRelayCLOSE := TRUE;
        T_OPENREQ(IN:=TRUE, PT:=T#1S);
        IF T_OPENREQ.Q THEN
            T_OPENREQ(IN:=FALSE);   // Reset Timer
            State := E_ShutterState.OPENTOGGLE;
        END_IF;
    END_IF
    *)

E_ShutterState.OPENTOGGLE :
    IF GVL_IO.bAmphosShutterCMD AND ShutterState
        THEN
        GVL_IO.bAmphosRelayCLOSE := TRUE;
        GVL_IO.bAmphosRelayOPEN := TRUE;
        T_OPENTOG(IN:=TRUE, PT:=T#1S);
        IF T_OPENTOG.Q THEN
            T_OPENTOG(IN:=FALSE);   // Reset Timer
            State := E_ShutterState.OPENACK;
        END_IF;
    END_IF

E_ShutterState.OPENACK :
    IF GVL_IO.bAmphosOn THEN
    GVL_IO.bAmphosRelayCLOSE := TRUE;
    GVL_IO.bAmphosRelayOPEN := TRUE;
        IF (NOT GVL_IO.bAmphosLaserACK) THEN
        State := E_ShutterState.OPENREADY;
        END_IF
    ELSE
    State := E_ShutterState.AMPHOSOFF;
    END_IF
(*
    IF GVL_IO.bAmphosShutterCMD AND LaserAck
    THEN
        State := E_ShutterState.OPENREADY;
    END_IF
    *)

E_ShutterState.OPENREADY :
    IF GVL_IO.bAmphosOn THEN
        IF (NOT GVL_IO.bAmphosLaserBusy) THEN
        State := E_ShutterState.OPENED;
        END_IF
    ELSE
    State := E_ShutterState.AMPHOSOFF;
    END_IF
(*
    IF GVL_IO.bAmphosShutterCMD AND (NOT LaserBusy) AND (NOT LaserAck)
        THEN
        State := E_ShutterState.OPENED;
    END_IF
*)
E_ShutterState.OPENED :
    IF GVL_IO.bAmphosOn THEN
        IF (NOT GVL_IO.bAmphosShutterCMD) THEN
            State := E_ShutterState.CLOSEREQ;
        END_IF
    ELSIF (NOT ShutterState) THEN
            State := E_ShutterState.CLOSEREQ;
    ELSE
    State := E_ShutterState.AMPHOSOFF;
    END_IF

E_ShutterState.CLOSEREQ :
    IF GVL_IO.bAmphosOn THEN
    GVL_IO.bAmphosRelayCLOSE := FALSE;
    GVL_IO.bAmphosRelayOPEN := TRUE;
        IF GVL_IO.bAmphosLaserACK OR (ShutterState) THEN
        State := E_ShutterState.CLOSEACK;
        END_IF
    ELSE
    State := E_ShutterState.AMPHOSOFF;
    END_IF
(*
    IF (NOT GVL_IO.bAmphosShutterCMD) AND (NOT ShutterState) AND (NOT LaserON) AND (LaserBusy)
        THEN
        GVL_IO.bAmphosRelayCLOSE := FALSE;
        GVL_IO.bAmphosRelayOPEN := TRUE;
        T_CLOSEREQ(IN:=TRUE, PT:=T#1S);
        IF T_CLOSEREQ.Q THEN
            T_CLOSEREQ(IN:=FALSE);   // Reset Timer
            State := E_ShutterState.CLOSETOGGLE;
        END_IF;
    END_IF
    *)

E_ShutterState.CLOSETOGGLE :
    IF (NOT GVL_IO.bAmphosShutterCMD) AND (NOT ShutterState)
        THEN
        GVL_IO.bAmphosRelayCLOSE := TRUE;
        GVL_IO.bAmphosRelayOPEN := TRUE;
        T_CLOSETOG(IN:=TRUE, PT:=T#1S);
        IF T_CLOSETOG.Q THEN
            T_CLOSETOG(IN:=FALSE);   // Reset Timer
            State := E_ShutterState.CLOSEACK;
        END_IF;
    END_IF

E_ShutterState.CLOSEACK :
    IF GVL_IO.bAmphosOn THEN
    GVL_IO.bAmphosRelayCLOSE := TRUE;
    GVL_IO.bAmphosRelayOPEN := TRUE;
        IF (NOT GVL_IO.bAmphosLaserACK) THEN
        State := E_ShutterState.CLOSEREADY;
        END_IF
    ELSE
    State := E_ShutterState.AMPHOSOFF;
    END_IF
(*
    IF (NOT GVL_IO.bAmphosShutterCMD) AND (NOT LaserAck)
        THEN
        State := E_ShutterState.CLOSEREADY;
    END_IF
*)

E_ShutterState.CLOSEREADY :
    IF GVL_IO.bAmphosOn THEN
        IF (NOT GVL_IO.bAmphosLaserBusy) THEN
        State := E_ShutterState.CLOSED;
        END_IF
    ELSE
    State := E_ShutterState.AMPHOSOFF;
    END_IF
(*
    IF (NOT GVL_IO.bAmphosShutterCMD) AND LaserBusy AND LaserAck
        THEN
        State := E_ShutterState.CLOSED;
    END_IF
    *)

E_ShutterState.CLOSED :
    IF GVL_IO.bAmphosOn THEN
        IF GVL_IO.bAmphosShutterCMD THEN
            State := E_ShutterState.OPENREQ;
        END_IF
    ELSIF (ShutterState) THEN
        State := E_ShutterState.OPENREQ;
    ELSE
    State := E_ShutterState.AMPHOSOFF;
    END_IF
END_CASE

END_FUNCTION_BLOCK

// ---- POUs/Devices/FB_LaserInterlock.TcPOU
FUNCTION_BLOCK FB_LaserInterlock
VAR_INPUT
    //bAmphosOn : BOOL; // Whether the amphos is on
    fOpcpaVoltage       : LREAL; // The voltage of the OPCPA
    fAmphosVoltage      : LREAL; // The Amphos voltage
    fMPCVoltage         : LREAL; // The MPC voltage
    AmphosStatus        : BOOL; //Amphos Laser Shutter Status
    bLoopTempOverride01 : BOOL; // Whether the chiller loop error is overriden
    bLoopTempOverride02 : BOOL; // Whether the chiller loop error is overriden
    bLoopTempOverride03 : BOOL; // Whether the chiller loop error is overriden
    bLoopTempOverride04 : BOOL; // Whether the chiller loop error is overriden
    bLoopTempOverride05 : BOOL; // Whether the chiller loop error is overriden
//    bShutterStatus      : BOOL; // Shutter Status
END_VAR

VAR_IN_OUT CONSTANT
    stErrors            : ST_ErrorStates; // Currently detected errors
    stOpcpaSetpoints    : ST_LaserSetpoints; // OPCPA setpoints
    stAmphosSetpoints   : ST_LaserSetpoints; // The Amphos setpoints
    stMPCSetpoints      : ST_LaserSetpoints; // The MPC setpoints
END_VAR

VAR_IN_OUT
    Mode              : E_Mode; // Mode
    bAmphosShutter   : BOOL; // Allowed Amphos Shutter state, point to NC Relay GVL
END_VAR

VAR
    bChillerErrors      : BOOL; // Local logical sum of chiller error states
    bTempSwitchErrors   : BOOL; // Local logical sum of temperature switch errors
    bAmphosUnderVolt    : BOOL; // Local var for checking Amphos under MinVoltage
    bOpcpaUnderVolt     : BOOL; // Local var for checking OPCPA under MinVoltage
    bMpcUnderVolt       : BOOL; // Local var for checking MPC under MinVoltage
END_VAR

VAR_OUTPUT
    bCarbideShutter  : BOOL; // Allowed Carbide Shutter state, point to NC Relay GVL
END_VAR

(*
The Amphos Shutter Enable function sends and Enable or Disable bit as an output to be used by the Amphos Shutter Command block
AmphosShutterEnable := TRUE := OPEN SHUTTER
AmphosShutterEnable := FALSE := CLOSE SHUTTER

Note : In master override modes, the Shutter state will hold the previous state value, unless manually forced
GVL_IO.bAmphosShutterEnable is the manual override PV for the shutter enable
*)

bChillerErrors := (
                 (NOT bLoopTempOverride01 AND stErrors.bChillerLoop01) OR
                 (NOT bLoopTempOverride02 AND stErrors.bChillerLoop02) OR
                 (NOT bLoopTempOverride03 AND stErrors.bChillerLoop03) OR
                 (NOT bLoopTempOverride04 AND stErrors.bChillerLoop04) OR
                 (NOT bLoopTempOverride05 AND stErrors.bChillerLoop05)
                 );
bTempSwitchErrors := (
                     NOT GVL_IO.bLoopTempSW01 OR
                     NOT GVL_IO.bLoopTempSW02 OR
                     NOT GVL_IO.bLoopTempSW03 OR
                     NOT GVL_IO.bLoopTempSW04 OR
                     NOT GVL_IO.bLoopTempSW05
                     );

bAmphosUnderVolt := fAmphosVoltage < stAmphosSetpoints.nMinVoltage;
bOpcpaUnderVolt := fOpcpaVoltage < stOpcpaSetpoints.nMinVoltage;
bMpcUnderVolt := fMPCVoltage < stMPCSetpoints.nMinVoltage;

CASE MODE OF
    // With great overrides comes great responsibility, and burnt optics
    E_Mode.MASTER_Override:
// Just pass and retain the previous Amphos Shutter State
//            bAmphosShutterIN := bAmphosShutterOUT;
        bCarbideShutter := TRUE;
        GVL_IO.bAmphosEnable := TRUE;
        bAmphosShutter := GVL_IO.bAmphosShutterEnable;

    E_Mode.Protection:
        // Close shutter if there is a hardware failure
        IF (stErrors.bHardwareFailure
        // Close shutter if there is a leak on the optical table with the amphos on, a leak under the table, or a leak inside the OPCPA with Carbide on
        (*OR stErrors.bLeakOpticalTableAmphosOn OR stErrors.bLeakOpcpaCarbideOn OR stErrors.bLeakUnderTable*)
        //Close shutter if the amphos is on and the temperature is too high in any loop. Ignore if operator override is enabled
         OR (bChillerErrors OR bTempSwitchErrors)
        // Close shutter if in OPCPA beam error state and OPCPA voltage too low
         OR (bOpcpaUnderVolt AND stErrors.bOpcpaBeam)
        // Close the shutter if there is a Dump Chiller error
         OR stErrors.bDumpChiller
        )
        // Check global IO for redundancy of Dump Chiller Errors
        OR (NOT GVL_IO.bDumpChillerFlow)
        OR (NOT GVL_IO.bBaseplateChillerFlow)
        THEN
            bAmphosShutter := bCarbideShutter := GVL_IO.bAmphosEnable := FALSE;
        ELSE
            // If the Amphos trips, always disable it
            IF bAmphosUnderVolt
            THEN
                //GVL_IO.bAmphosShutterEnable MUST be overwritten to update EPICS downstream
                bAmphosShutter := GVL_IO.bAmphosEnable := GVL_IO.bAmphosShutterEnable:= FALSE;
            ELSE
                bAmphosShutter := GVL_IO.bAmphosEnable := TRUE;
            END_IF
            // Only open the Amphos shutter if all 3 lasers are happy
            IF (NOT(bAmphosUnderVolt OR bOpcpaUnderVolt OR bMpcUnderVolt))
            THEN
                //GVL_IO.bAmphosShutterEnable MUST be overwritten to update EPICS downstream
                bAmphosShutter := GVL_IO.bAmphosShutterEnable:= TRUE;
            ELSE
                //GVL_IO.bAmphosShutterEnable MUST be overwritten to update EPICS downstream
                bAmphosShutter := GVL_IO.bAmphosShutterEnable:= FALSE;
            END_IF
            // Carbide Shutter is weird, allows solo Carbide use explicitly
            IF NOT (bAmphosUnderVolt OR bOpcpaUnderVolt OR bMpcUnderVolt)
                // This state is physically impossible
                OR (bAmphosUnderVolt AND NOT bOpcpaUnderVolt AND NOT bMpcUnderVolt)
                // But this state happens when the AMPHOS is powered down
                OR (bAmphosUnderVolt AND bOpcpaUnderVolt AND NOT bMpcUnderVolt)
            THEN
                bCarbideShutter := TRUE;
            ELSE
                bCarbideShutter := FALSE;
            END_IF
        END_IF

    E_Mode.AMPHOS_Maintenance:
    // Close shutter if there is a hardware failure
        IF (stErrors.bHardwareFailure
        // Close shutter if there is a leak on the optical table with the amphos on, a leak under the table, or a leak inside the OPCPA with Carbide on
        (*OR stErrors.bLeakOpticalTableAmphosOn OR stErrors.bLeakOpcpaCarbideOn OR stErrors.bLeakUnderTable*)
        //Close shutter if the amphos is on and the temperature is too high in any loop. Ignore if operator override is enabled
         OR (bChillerErrors OR bTempSwitchErrors)
        // Close the shutter if there is a Dump Chiller error
         OR stErrors.bDumpChiller
        )
        // Check global IO for redundancy of Chiller Errors
        OR (NOT GVL_IO.bDumpChillerFlow)
        OR (NOT GVL_IO.bBaseplateChillerFlow)
        THEN
            //GVL_IO.bAmphosShutterEnable MUST be overwritten to update EPICS downstream
            bAmphosShutter := bCarbideShutter := GVL_IO.bAmphosEnable := FALSE;
        ELSE
    // Just pass the Amphos shutter state and keep it enabled
            GVL_IO.bAmphosEnable := TRUE;
            //GVL_IO.bAmphosShutterEnable MUST be overwritten to update EPICS downstream
            bAmphosShutter := GVL_IO.bAmphosShutterEnable;
        END_IF
    // Close the carbide shutter if the MPC is unhappy
    IF bMpcUnderVolt
    THEN
        bCarbideShutter := FALSE;
    ELSE
        bCarbideShutter := TRUE;
    END_IF

    // Undefined state, do not get here. Do not pass go, do not collect 200 dollars
    ELSE
    // If you get stuck here you deserve it
        Mode := E_Mode.Protection;
END_CASE

END_FUNCTION_BLOCK

// ---- POUs/Interlocks/F_DumpChillerEnable.TcPOU
// Interlock logic for the Dump Chiller
FUNCTION F_DumpChillerEnable : BOOL
VAR_INPUT
    //bMasterOverride : BOOL; //Master manual override control input
    Mode : E_Mode;
END_VAR
VAR_IN_OUT CONSTANT
    stErrors : ST_ErrorStates; // Currently detected errors
END_VAR
VAR
END_VAR

// Disable dump chiller if there's a hardware failure
IF (stErrors.bHardwareFailure
    // Disable dump chiller for these leak conditions
    //OR stErrors.bLeakOpticalTableAmphosOn OR stErrors.bLeakOpticalTableNoLaser OR stErrors.bLeakOpcpaCarbideOn OR stErrors.bLeakUnderTable)
   OR stErrors.bLeakUnderTable)
THEN
    F_DumpChillerEnable := FALSE;
ELSE
    CASE MODE OF
        E_Mode.MASTER_Override:
            F_DumpChillerEnable := TRUE;
        // Otherwise things are okay
        ELSE
            F_DumpChillerEnable := TRUE;
    END_CASE
END_IF

END_FUNCTION

// ---- POUs/Interlocks/F_BaseplateChillerEnable.TcPOU
// Interlock logic for the Baseplate Chiller
FUNCTION F_BaseplateChillerEnable : BOOL
VAR_INPUT
       //bMasterOverride : BOOL; //Master manual override control input
       Mode : E_Mode; // Mode of operation
END_VAR
VAR_IN_OUT CONSTANT
    stErrors : ST_ErrorStates; // Currently detected errors
END_VAR
VAR
END_VAR

// Disable baseplate chiller if there is a hardware failure or leak under the table
IF (stErrors.bHardwareFailure OR stErrors.bLeakUnderTable)
    THEN
    F_BasePlateChillerEnable := FALSE;
    ELSE
    CASE MODE OF
        // Master override does indeed override
        E_Mode.MASTER_Override:
           F_BasePlateChillerEnable := TRUE;
        // And yet redundantly our default state is TRUE?
        ELSE
           F_BasePlateChillerEnable := TRUE;
    END_CASE
END_IF

END_FUNCTION
